(* IEC 61131-3 sources: assembler/src, 6 files *)

(* ---- Clamp.st ---- *)
CLASS ClampBase
    VAR
        _baseAtPlace: REF_TO DiffuseSensor;
        _partLeaving: REF_TO DiffuseSensor;
        _baseClamped:BOOL;
        _clampBase: BOOL;
    END_VAR

    METHOD PUBLIC Init
        VAR_INPUT
            BaseAtPlace: REF_TO DiffuseSensor;
            PartLeaving: REF_TO DiffuseSensor;
        END_VAR
        _baseAtPlace := BaseAtPlace;
        _partLeaving := PartLeaving;
    END_METHOD

    METHOD PUBLIC IsObjectReached : BOOL
        IsObjectReached := _baseAtPlace^.IsObjectDetected();
    END_METHOD

    METHOD PUBLIC IsObjectLeft : BOOL
        IsObjectLeft := _partLeaving^.IsObjectDetected();
    END_METHOD

    METHOD PUBLIC IsObjectClamped : BOOL
        IsObjectClamped := _baseClamped;
    END_METHOD

    METHOD PUBLIC ClampObject
        _clampBase := TRUE;
    END_METHOD

    METHOD PUBLIC Execute
        VAR_INPUT
            baseClamped: BOOL;
        END_VAR
        VAR_OUTPUT
            clampBase: BOOL;
        END_VAR

        _baseClamped := baseClamped;

        IF(THIS.IsObjectReached()) THEN
            THIS.ClampObject();
        END_IF;

        clampBase := _clampBase;
    END_METHOD
END_CLASS

(* ---- Conveyor.st ---- *)
CLASS Conveyor
    VAR
        _started: BOOL;
    END_VAR

    METHOD PUBLIC Start
        _started := TRUE;
    END_METHOD

    METHOD PUBLIC Stop
        _started := FALSE;
    END_METHOD

    METHOD PUBLIC Execute
        VAR_OUTPUT
            output: BOOL;
        END_VAR
        output := _started;
    END_METHOD
END_CLASS

(* ---- DiffuseSensor.st ---- *)
CLASS DiffuseSensor
    VAR
        _input : BOOL;
    END_VAR

    METHOD PUBLIC IsObjectDetected : BOOL
        IsObjectDetected := NOT _input;
    END_METHOD

    METHOD PUBLIC Execute
        VAR_INPUT
            input : BOOL;
        END_VAR
        _input := input;
    END_METHOD
END_CLASS

(* ---- configuration.st ---- *)
USING Siemens.Simatic.S71500.Tasks;

TYPE
    MachineStatus: (NotStarted, Started, Stopped);
END_TYPE

CONFIGURATION MyConfiguration
    TASK MyProgramCycleTask : Siemens.Simatic.S71500.Tasks.ProgramCycle;
    PROGRAM MyCyclicProgram WITH MyProgramCycleTask : MyProgram;

    TASK MyStartupTask : Startup;
    PROGRAM MyStartupProgram WITH MyStartupTask : LoadConfiguration;

    VAR_GLOBAL
        MovingXInput AT %I0.0: BOOL;
        MovingZInput AT %I0.1: BOOL;
        ItemDetectedInput AT %I0.2: BOOL;
        LidAtPlaceInput AT %I0.3: BOOL;
        LidClampedInput AT %I0.4: BOOL;
        PosAtLimitLidsInput AT %I0.5: BOOL;
        BaseAtPlaceInput AT %I0.6: BOOL;
        BaseClampedInput AT %I0.7: BOOL;
        PosAtLimitBasesInput AT %I1.0: BOOL;
        PartLeavingInput AT %I1.1: BOOL;
        StartInput AT %I1.2: BOOL;
        ResetInput AT %I1.3: BOOL;
        StopInput AT %I1.4: BOOL;
        EmergencyStopInput AT %I1.5: BOOL;
        AutoInput AT %I1.6: BOOL;
        FactoryIORunningInput AT %I1.7: BOOL;
        MoveXOutput AT %Q0.0: BOOL;
        MoveZOutput AT %Q0.1: BOOL;
        GrabOutput AT %Q0.2: BOOL;
        LidsConveyorOutput AT %Q0.3: BOOL;
        ClampLidOutput AT %Q0.4: BOOL;
        PosRaiseLidsOutput AT %Q0.5: BOOL;
        BasesConveyorOutput AT %Q0.6: BOOL;
        ClampBaseOutput AT %Q0.7: BOOL;
        PosRaiseBasesOutput AT %Q1.0: BOOL;
        StartLightOutput AT %Q1.1: BOOL;
        ResetLightOutput AT %Q1.2: BOOL;
        StopLightOutput AT %Q1.3: BOOL;
        CounterOutput AT %QD30: DINT;
    END_VAR

    VAR_GLOBAL
        BasesConveyor : Conveyor;
        LidsConveyor : Conveyor;
        ClampBase: ClampBase;
        BaseAtPlace: DiffuseSensor;
        PartLeaving: DiffuseSensor;

        MachineStatus: MachineStatus;
    END_VAR
END_CONFIGURATION

(* ---- InitProgram.st ---- *)
PROGRAM LoadConfiguration
    VAR_EXTERNAL
        BasesConveyor : Conveyor;
        LidsConveyor : Conveyor;
        ClampBase: ClampBase;
        BaseAtPlace: DiffuseSensor;
        PartLeaving: DiffuseSensor;

        LidsConveyorOutput : BOOL;
        BasesConveyorOutput : BOOL;
    END_VAR

    ClampBase.Init(REF(BaseAtPlace), REF(PartLeaving));
    BasesConveyor.Stop();
    LidsConveyor.Stop();
END_PROGRAM

(* ---- program.st ---- *)
PROGRAM MyProgram
    VAR_EXTERNAL
        MovingXInput : BOOL;
        MovingZInput : BOOL;
        ItemDetectedInput : BOOL;
        LidAtPlaceInput : BOOL;
        LidClampedInput : BOOL;
        PosAtLimitLidsInput : BOOL;
        BaseAtPlaceInput : BOOL;
        BaseClampedInput : BOOL;
        PosAtLimitBasesInput : BOOL;
        PartLeavingInput : BOOL;
        StartInput : BOOL;
        ResetInput : BOOL;
        StopInput : BOOL;
        EmergencyStopInput : BOOL;
        AutoInput : BOOL;
        FactoryIORunningInput : BOOL;
        MoveXOutput : BOOL;
        MoveZOutput : BOOL;
        GrabOutput : BOOL;
        LidsConveyorOutput : BOOL;
        ClampLidOutput : BOOL;
        PosRaiseLidsOutput : BOOL;
        BasesConveyorOutput : BOOL;
        ClampBaseOutput : BOOL;
        PosRaiseBasesOutput : BOOL;
        StartLightOutput : BOOL;
        ResetLightOutput : BOOL;
        StopLightOutput : BOOL;
        CounterOutput : DINT;
        BasesConveyor : Conveyor;
        LidsConveyor : Conveyor;
        ClampBase : ClampBase;
        BaseAtPlace : DiffuseSensor;
        PartLeaving : DiffuseSensor;
        MachineStatus : MachineStatus;
    END_VAR
    CyclicIO();

    IF StartInput THEN
        StartLightOutput := TRUE;
        MachineStatus := MachineStatus#Started;
    ELSE
        StartLightOutput := FALSE;
    END_IF;

    IF NOT(StopInput) THEN
        StopLightOutput := TRUE;
        MachineStatus := MachineStatus#Stopped;
    ELSE
        StopLightOutput := FALSE;
    END_IF;

    CASE MachineStatus OF
        MachineStatus#NotStarted:
            ;
        MachineStatus#Started:
            BasesConveyor.Start();
            LidsConveyor.Start();
        MachineStatus#Stopped:
            BasesConveyor.Stop();
            LidsConveyor.Stop();
    END_CASE;

    BasesConveyor.Execute(BasesConveyorOutput);
    LidsConveyor.Execute(LidsConveyorOutput);
END_PROGRAM
